{attribute addProperty BoxType "EK1100-0000-0018"}
{attribute addProperty Id "Beckhoff_EP9xxxEK1122Beckhoff_EP9xxxEK1122_888C15454760595A_0023_EP9224_1037_0017EP9224_179A0949162A_0015_EP9128_2021_0019EP9128_179A0949162A_0014_EP9128_1021_0019EP9128_179A0949162A_0012_EP9128_2021_0018EP9128_179A0949162A_0011_EP9128_1021_0018EP9128_179A0949162A_0009_EP9128_2021_0017EP9128_179A0949162A_0008_EP9128_1021_0017EP9128_179A0949162A_0006_EP9128_2021_0016EP9128_179A0949162A_0005_EP9128_1021_0016EP9128_179A0949162A_0003_EP9128_2020_0016EP9128_179A0949162A_0002_EP9128_1020_0016EP9128_179A0949162"}
{attribute addProperty CRC "3006303804"}
{attribute addProperty SizeInBites "4936"}
{attribute addProperty SizeInBytes "617"}
TYPE Beckhoff_EP9xxx_B3308E3C EXTENDS EK1100_179A0949 :
STRUCT
	{attribute addProperty Name "Beckhoff_EP9xxxEK1122"}
	Beckhoff_EP9xxxEK1122 : Beckhoff_EP9xxxEK1122_888C1545;
	{attribute addProperty Name "A_0023_EP9224_1037_0017"}
	A_0023_EP9224_1037_0017 : EP9224_179A0949;
	{attribute addProperty Name "A_0015_EP9128_2021_0019"}
	A_0015_EP9128_2021_0019 : EP9128_179A0949;
	{attribute addProperty Name "A_0014_EP9128_1021_0019"}
	A_0014_EP9128_1021_0019 : EP9128_179A0949;
	{attribute addProperty Name "A_0012_EP9128_2021_0018"}
	A_0012_EP9128_2021_0018 : EP9128_179A0949;
	{attribute addProperty Name "A_0011_EP9128_1021_0018"}
	A_0011_EP9128_1021_0018 : EP9128_179A0949;
	{attribute addProperty Name "A_0009_EP9128_2021_0017"}
	A_0009_EP9128_2021_0017 : EP9128_179A0949;
	{attribute addProperty Name "A_0008_EP9128_1021_0017"}
	A_0008_EP9128_1021_0017 : EP9128_179A0949;
	{attribute addProperty Name "A_0006_EP9128_2021_0016"}
	A_0006_EP9128_2021_0016 : EP9128_179A0949;
	{attribute addProperty Name "A_0005_EP9128_1021_0016"}
	A_0005_EP9128_1021_0016 : EP9128_179A0949;
	{attribute addProperty Name "A_0003_EP9128_2020_0016"}
	A_0003_EP9128_2020_0016 : EP9128_179A0949;
	{attribute addProperty Name "A_0002_EP9128_1020_0016"}
	A_0002_EP9128_1020_0016 : EP9128_179A0949;
END_STRUCT
END_TYPE

(* stored: Version 1.2.0.0, ProductVersion 3.1.4024.9
   DUT Beckhoff_EP9xxx_B3308E3C: Id {79a74cd2-26b1-465f-a381-86e1111fa889} *)
